Staubli VAL3: goHome.pgx

program goHome(num& x_nMoveID (dimensions=1))
  local num l_nError
  local num l_nTrackStatus
begin
  // This program sends the robot to the jHome position. If the
  //  robot is synchronized with a conveyor, the program uses a
  //  de-synchronization move instruction, otherwise the program
  //  uses a standard move instruction.
  //
  // Input parameters
  //  None            :
  //
  // Output parameters
  //  x_nMoveID       : Motion stack ID for this move
  //
  //----------------------------------------------------------------
  //
  _bSentToHome=true
  //
  call mot:getTrackStatus(l_nTrackStatus)
  if l_nTrackStatus>0
    // Use trackOff if the robot is synchronized
    call mot:trackOffJ(jHome,tGripper,mNomSpeed,x_nMoveID,l_nError)
  else
    // Use movej if the robot is not synchronized
    x_nMoveID=movej(jHome,tGripper,mNomSpeed)
  endIf
  //
end
